Fanuc KAREL source: kt00476.KL

-- PROVISIONAL review KL for V1013-1; original PC SHA256 53b54c54b41822f4c82dadcc9fbbb5118aeb01be447911a290ff6b742d0a804b
-- Incomplete behavior may be omitted. Consult companion uncertainty JSON. Do not deploy.
PROGRAM KT00476
%NOLOCKGROUP
-- UNRESOLVED_DECL P1 type=000101
-- UNRESOLVED_DECL P2 type=000101
-- UNRESOLVED_DECL OUT type=000106
BEGIN
  -- UNRESOLVED_PC offsets 5-34; opcodes 49,49,60,7E,4A
  -- UNRESOLVED_PC offsets 39-43; opcodes 7F
END KT00476
